FUNCTION_BLOCK Scharr (* openCV scharr filter *)
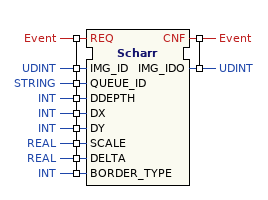
  EVENT_INPUT
    REQ WITH IMG_ID, QUEUE_ID, DDEPTH, DX, DY, SCALE, DELTA, BORDER_TYPE;
  END_EVENT
  EVENT_OUTPUT
    CNF WITH IMG_IDO;
  END_EVENT
  VAR_INPUT
    IMG_ID : UDINT;
    QUEUE_ID : STRING;
    DDEPTH : INT;
    DX : INT;
    DY : INT;
    SCALE : REAL;
    DELTA : REAL;
    BORDER_TYPE : INT;
  END_VAR
  VAR_OUTPUT
    IMG_IDO : UDINT;
  END_VAR
END_FUNCTION_BLOCK
(* other elements stored in the file *)
(* morphologyDefaultBorderValue *)
